Yaskawa INFORM job: 2-YMP.JBI

/JOB
//NAME 2-YMP
///FOLDERNAME INNE
//POS
///NPOS 2,2,0,0,0,0
///TOOL 0
///POSTYPE PULSE
///PULSE
C00000=-106109,30553,56766,-22429,74075,-32630
C00001=107812,67577,98417,23313,67808,32740
BC00000=277960,863803,688929
BC00001=277960,1283097,688929
//INST
///DATE 2023/10/04 15:13
///ATTR SC,RW
///GROUP1 RB1,BS1
NOP
MOVJ C00000 BC00000 VJ=0.78
MOVJ C00001 BC00001 VJ=0.78
END
